FUNCTION_BLOCK TcoTixonPickVibro_v_1_x_x EXTENDS TcoCore.TcoComponent

VAR_INPUT
	inControllerInAuto  : BOOL;
	inNotEmptyFeeder  : BOOL;	
	inSeparatorHomePos  : BOOL;
	inFillingSensor  : BOOL; 
	inSeparatorPresent  : BOOL;
	inSeparatorWorkPos  : BOOL;
	inPickZone  : BOOL;
END_VAR
VAR_OUTPUT
	outFeedingA : BOOL;
	outSepareComponent : BOOL;
	outBlowValveA : BOOL;
	outRedLed : BOOL;	
	outGreenLed : BOOL;
	outHopper : BOOL;
	outFeedingB : BOOL;
	outBlowValveB : BOOL;
	
END_VAR
VAR

    {attribute addProperty Name "<#Status#>"}
    {attribute clr [ReadOnly()]}
    _status : TcoTixonPickVibro_Status_v_1_x_x;
    {attribute addProperty Name "<#Control#>"}
    _control : TcoTixonPickVibro_Control_v_1_x_x;
    {attribute addProperty Name "<#Config#>"}
    _config : TcoTixonPickVibro_Config_v_1_x_x;

    _someTaskIsActive : BOOL;

    {attribute 'hide'}
    _blink : TcoUtilities.TcoBlinker(THIS^);
    _runAutomatic : BOOL;
    _hasError : BOOL;
END_VAR
VAR

    {attribute addProperty Name "<#Separator task#>"}
    _separatorTask : TcoTixonPickVibroSeparatorTask(THIS^);
    {attribute addProperty Name "<#Buffer task#>"}
    _bufferTask : TcoTixonBufferTask(THIS^);
    {attribute addProperty Name "<#Vibrating bin task#>"}
    _binFeederTask : TcoTixonPickVibroFeederTask(THIS^);
    {attribute addProperty Name "<#Hopper task#>"}
    _hopperTask : TcoTixonHopperTask(THIS^);

    {attribute addProperty Name "<#Restore#>"}
    _restoreTask : TcoCore.TcoTask(THIS^);

END_VAR

VAR
    {attribute 'hide'}
    _sb : TcoCore.StringBuilder;
END_VAR



_blink(inOnTime:=_config.BlinkTime,inOffTime:=_config.BlinkTime);		
UpdateStatus();

_separatorTask.Enabled:=TRUE;
_separatorTask(inoConfig:=_config,inoControl:=_control,inoStatus:=_status);
_bufferTask.Enabled:=TRUE;
_bufferTask(inoConfig:=_config,inoControl:=_control,inoStatus:=_status);
_binFeederTask.Enabled:=TRUE;
_binFeederTask(inoConfig:=_config,inoControl:=_control,inoStatus:=_status);
_hopperTask.Enabled := _config.HopperActive;
_hopperTask(inoConfig:=_config,inoControl:=_control,inoStatus:=_status);







//*************RESTORE********************

_restoreTask.Enabled := TRUE;
IF _restoreTask.Execute() THEN
	Restore();
	_restoreTask.DoneWhen(TRUE);
END_IF
//****************************************


UpdateControl();

METHOD PUBLIC BufferFeed : TcoCore.ITcoTaskStatus
BufferFeed:=_bufferTask.Invoke();
_bufferTask.AutoRestore:=false;
END_METHOD

PROPERTY PUBLIC BufferTask : REFERENCE TO TcoTixonBufferTask
GET
BufferTask ref= _bufferTask;
END_GET
END_PROPERTY

(*~
	<docu>
		<summary>
			Gets the configuration of the Tixon Step. 					
		</summary>			
	</docu>	
~*)
PROPERTY Config : REFERENCE TO TcoTixonPickVibro_Config_v_1_x_x
GET
Config REF= _config;
END_GET
END_PROPERTY

METHOD PUBLIC CyclicBinFeed : TcoCore.ITcoTaskStatus
VAR_INPUT
END_VAR
CyclicBinFeed:=_binFeederTask.Invoke();
_binFeederTask.AutoRestore:=true;
END_METHOD

METHOD PUBLIC CyclicBufferFeed : TcoCore.ITcoTaskStatus
CyclicBufferFeed:=_bufferTask.Invoke();
_bufferTask.AutoRestore:=true;
END_METHOD

METHOD PUBLIC CyclicHopperFeed : TcoCore.ITcoTaskStatus
CyclicHopperFeed:=_hopperTask.Invoke();
_hopperTask.AutoRestore:=TRUE;
END_METHOD

METHOD PUBLIC CyclicSepare : TcoCore.ITcoTaskStatus
CyclicSepare:=_separatorTask.Invoke();
_separatorTask.AutoRestore:=true;
END_METHOD

METHOD PUBLIC DefaultSignalisation
VAR_INPUT
END_VAR
// led signalisation
_hasError:=_separatorTask.Error OR _bufferTask.Error OR _hopperTask.Error;
_control.GreenLed:=FALSE;
_control.RedLed:=FALSE;
IF  NOT _status.ControllerInAuto  THEN
	_control.GreenLed:=TRUE;
	_control.RedLed:=TRUE;
ELSIF _hasError AND _blink.IsOn  AND _status.ControllerInAuto  THEN
	_control.RedLed:=TRUE;
ELSIF _status.ControllerInAuto AND NOT _hasError AND _status.NotEmptyFeeder THEN
	_control.GreenLed:=TRUE;
ELSIF _blink.IsOn AND _status.ControllerInAuto AND NOT _status.NotEmptyFeeder THEN
	_control.GreenLed:=TRUE;
	_control.RedLed:=TRUE;
END_IF
END_METHOD

METHOD PUBLIC HopperFeed : TcoCore.ITcoTaskStatus
HopperFeed:=_hopperTask.Invoke();
_hopperTask.AutoRestore:=false;
END_METHOD

PROPERTY PUBLIC HopperTask : reference TO TcoTixonHopperTask
GET
HopperTask ref= _hopperTask;
END_GET
END_PROPERTY

(*~
	<docu>
		<summary>
			Restores this instance to the Ready state. Can be called explicitly or from within one of the restore mechanisms.	
		</summary>			
	</docu>	
~*)
METHOD Restore : ITcoRestorable
RestoreTasks();
_control.BlowAValve:=FALSE;
_control.FeedingA:=FALSE;
_control.GreenLed:=FALSE;
_control.RedLed:=FALSE;
_control.SepareComponent:=FALSE;
_control.FeedingB:=FALSE;
_control.BlowValveB:=FALSE;
_control.Hooper:=FALSE;
END_METHOD

METHOD INTERNAL RestoreTasks
//_resetTask.Restore();

_separatorTask.Restore();
_bufferTask.Restore();
_binFeederTask.Restore();
_hopperTask.Restore();
END_METHOD

PROPERTY PUBLIC SeparatorTask : REFERENCE TO TcoTixonPickVibroSeparatorTask
GET
SeparatorTask ref= _separatorTask;
END_GET
END_PROPERTY

METHOD PUBLIC Separe : TcoCore.ITcoTaskStatus
Separe:=_separatorTask.Invoke();
_separatorTask.AutoRestore:=false;
END_METHOD

(*~
	<docu>
		<summary>
		    Custom service (manual, maintenance) logic.
			This method must be implemented in derived class.
		</summary>			
	</docu>	
~*)
METHOD PROTECTED ServiceMode
END_METHOD

(*~
	<docu>
		<summary>
			Gets the status of the Tixon Step. 					
		</summary>			
	</docu>	
~*)
PROPERTY Status : REFERENCE TO TcoTixonPickVibro_Status_v_1_x_x
GET
Status REF= _status;
END_GET
END_PROPERTY

METHOD INTERNAL UpdateControl
VAR_INPUT
END_VAR

VAR
	index: INT;
END_VAR
outBlowValveA:= _control.BlowAValve;
outFeedingA:=_control.FeedingA;
outGreenLed:=_control.GreenLed;
outRedLed:=_control.RedLed;
outSepareComponent:=_control.SepareComponent;
outFeedingB:=_control.FeedingB;
outBlowValveB:=_control.BlowValveB;
outHopper:=_control.Hooper;
END_METHOD

METHOD INTERNAL UpdateStatus
VAR
    
END_VAR
_status.NotEmptyFeeder:=inNotEmptyFeeder;
_status.FillingSensor:=inFillingSensor;
_status.SeparatorHomePos:=inSeparatorHomePos;
_status.SeparatorPresent:=inSeparatorPresent;
_status.SeparatorWorkPos:=inSeparatorWorkPos;
_status.ControllerInAuto:=inControllerInAuto;
_status.InPickZone:=inPickZone;
END_METHOD

END_FUNCTION_BLOCK

(* stored: Version 1.1.0.1, ProductVersion 3.1.4024.12
   POU TcoTixonPickVibro_v_1_x_x: Id {5d44d987-7de3-03df-09ae-c764cdfb8d80}, SpecialFunc None
   Folder Operations: Id {915c5c8c-e4ad-0edb-2d19-f83ce84fee09}
   Folder Loop: Id {fbffec73-29f7-0f61-12da-62aed55d6d93}
   Folder Single: Id {31401d1b-fbb9-0d0e-25cd-b2f0eb368e0d}
   Folder Task: Id {6f2723cb-27ef-09a0-07e6-b81c88868551}
   Method BufferFeed: Id {9390702e-fa93-0e1e-06d9-a1953b5d43df}
   Property BufferTask: Id {ab88bcb3-a0b1-0295-2445-c33abff0f050}
   Get Get: Id {a6643d15-ccdb-0356-39f4-30a639398a41}
   Property Config: Id {bac766df-24ab-0afe-0792-40e103ff5fab}
   Get Get: Id {d32e8b23-6375-0cd3-1dbb-693d99a0f330}
   Method CyclicBinFeed: Id {9e7b8238-ac0f-0fe0-3778-9a33e96392c7}
   Method CyclicBufferFeed: Id {e60f056d-2901-0b7a-0673-1ad36a68068e}
   Method CyclicHopperFeed: Id {7770a31b-0cfa-0466-2f62-4698af32dfc2}
   Method CyclicSepare: Id {a2ffd8d6-d9a3-0581-3b53-3172f7b503b3}
   Method DefaultSignalisation: Id {ce8c6dc9-946a-0ae7-1123-2d7dd2f48087}
   Method HopperFeed: Id {10ce520c-37cb-05fa-05d0-09d37e6f4cb0}
   Property HopperTask: Id {5cf54943-9c5b-0c22-10ef-277f2fa1254d}
   Get Get: Id {6fe43ffc-9cd5-0abb-13fb-e00cd6427080}
   Method Restore: Id {8644f063-a070-0375-0bdb-3c8072e80800}
   Method RestoreTasks: Id {370e966c-9a70-0709-2cf0-2eee25ceb8ad}
   Property SeparatorTask: Id {b82d4086-3a66-07c8-099c-4570d40f25ab}
   Get Get: Id {8dc9ac57-b141-0b7f-0db3-2a56556bae1c}
   Method Separe: Id {f4a12d2f-a6d1-05fa-1cfd-29e32305e394}
   Method ServiceMode: Id {5df3361d-135f-0f46-35a7-90714454738f}
   Property Status: Id {7a4a5ce4-ae4a-0efa-0f3f-915619140643}
   Get Get: Id {e24c715d-151c-082c-186d-2839c9092ffc}
   Method UpdateControl: Id {28bc6cd8-fcf0-0c04-1762-c17c9b5f533b}
   Method UpdateStatus: Id {72ad5663-eb66-0d5e-1067-946942f56894} *)
